FUNCTION FC_GetLocalTimeStringMinAccuracy : T_SHORT_STR	// Returns the local time as short string, eg. '08:02 AM'.
													// Use E_REGIO_SELECTION at FB_CycleStart for a different format.

FC_GetLocalTimeStringMinAccuracy := IING.localTimeMinAccuracy;

END_FUNCTION

(* stored: Version 1.1.0.1, ProductVersion 3.1.4026.18
   POU FC_GetLocalTimeStringMinAccuracy: Id {396b1c6b-b1f5-44d4-9835-57f39def515d}, SpecialFunc None *)
